PROGRAM sonotecCalibration
VAR_INPUT
	start : BOOL := FALSE;
	pumpA : BOOL := TRUE;
	setSpeedDuration : TIME := T#2M;
	runTestDuration : TIME := T#5M;
END_VAR
VAR_OUTPUT
	results : ARRAY[1..50] OF testResults;
END_VAR
VAR
	i : UINT := 0; // index
	n : UINT := 7;
	t : LREAL := 0.0;
	sp : ARRAY [1..50] OF LREAL := [80.0, 160.0, 240.0, 320.0, 400.0, 480.0, 560.0];
	//sp : ARRAY [1..50] OF LREAL := [51.0, 58.0, 64.0, 79.0, 97.0, 112.0, 128.0, 151.0, 210.0, 280.0, 335.0, 410.0, 480.0, 600.0];
	//sp : ARRAY [1..50] OF LREAL := [335.0, 410.0, 480.0, 600.0];
	setSpeed : SFCStepType;
	runTest : SFCStepType;
	recordTest : SFCStepType;
END_VAR

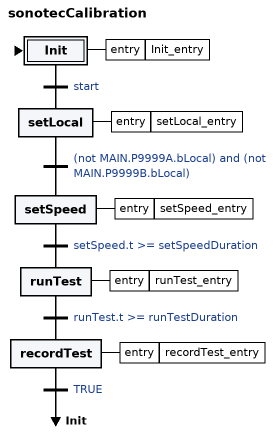
INITIAL_STEP Init:
    Init_entry(P1);  // entry action
END_STEP
TRANSITION FROM Init TO setLocal
    := start;
END_TRANSITION
STEP setLocal:
    setLocal_entry(P1);  // entry action
END_STEP
TRANSITION FROM setLocal TO setSpeed
    := (not MAIN.P9999A.bLocal) and (not MAIN.P9999B.bLocal);
END_TRANSITION
STEP setSpeed:
    setSpeed_entry(P1);  // entry action
END_STEP
TRANSITION FROM setSpeed TO runTest
    := setSpeed.t >= setSpeedDuration;
END_TRANSITION
STEP runTest:
    runTest_entry(P1);  // entry action
END_STEP
TRANSITION FROM runTest TO recordTest
    := runTest.t >= runTestDuration;
END_TRANSITION
STEP recordTest:
    recordTest_entry(P1);  // entry action
END_STEP
TRANSITION FROM recordTest TO Init
    := TRUE;
END_TRANSITION

ACTION setLocal_entry:
IF MAIN.P9999A.bLocal THEN
	MAIN.P9999A.nLocal_RQ := 0;  //put pump in remote
END_IF
IF MAIN.P9999B.bLocal THEN
	MAIN.P9999B.nLocal_RQ := 0;  //put pump in remote
END_IF
END_ACTION

ACTION runTest_entry:
MAIN.fbFQ9999A.resetRQ := TRUE;
MAIN.fbFQ9999B.resetRQ := TRUE;
MAIN.fbFQ9999C.resetRQ := TRUE;
END_ACTION

ACTION setSpeed_entry:
i := i + 1;
results[i].FQ9999A := 0.0;
results[i].FQ9999B := 0.0;
results[i].FQ9999C := 0.0;
results[i].FT9999Aavg := 0.0;
results[i].FT9999Bavg := 0.0;
results[i].FT9999Cavg := 0.0;
IF pumpA THEN
	results[i].P9999Arpm := sp[i];
	results[i].P9999Brpm := 0.0;
	MAIN.P9999A.nRun_RQ := 1; //start pump
	MAIN.P9999A.fSpeedSP_RQ := sp[i];
	MAIN.P9999B.nRun_RQ := 0; //stop pump
	MAIN.P9999B.fSpeedSP_RQ := 0.0;
ELSE
	results[i].P9999Arpm := 0.0;
	results[i].P9999Brpm := sp[i];
	MAIN.P9999A.nRun_RQ := 0; //stop pump
	MAIN.P9999A.fSpeedSP_RQ := 0.0;
	MAIN.P9999B.nRun_RQ := 1; //start pump
	MAIN.P9999B.fSpeedSP_RQ := sp[i];
END_IF
results[i].P9999Atubing := MAIN.P9999A.nTubeSize;
results[i].P9999Btubing := MAIN.P9999B.nTubeSize;
END_ACTION

ACTION recordTest_entry:
results[i].FQ9999A := MAIN.fbFQ9999A.total;
results[i].FQ9999B := MAIN.fbFQ9999B.total;
results[i].FQ9999C := MAIN.fbFQ9999C.total;
t := DWORD_TO_LREAL(TIME_TO_DWORD(runTestDuration))/1000.0/60.0;
results[i].FT9999Aavg := MAIN.fbFQ9999A.total/t;
results[i].FT9999Bavg := MAIN.fbFQ9999B.total/t;
results[i].FT9999Cavg := MAIN.fbFQ9999C.total/t;
END_ACTION

ACTION Init_entry:
IF i >= n THEN
	MAIN.P9999A.nRun_RQ := 0; //stop pump
	MAIN.P9999B.nRun_RQ := 0; //stop pump
	start := FALSE;
	i := 0;
END_IF
END_ACTION

END_PROGRAM

(* stored: Version 1.1.0.1, ProductVersion 3.1.0.36
   POU sonotecCalibration: Id {d8cace5d-4622-4721-8ad4-24bb2227c384}, SpecialFunc None
   Action setLocal_entry: Id {5f66cdec-b477-4613-901d-62d885f9dd8f}
   Action runTest_entry: Id {c408255e-879f-4b7c-a447-719d9549f349}
   Action setSpeed_entry: Id {d2f1a663-0229-4750-b307-3ef7969d2ce6}
   Action recordTest_entry: Id {ebcff068-10a2-4957-bb37-8ab7e3b316fc}
   Action Init_entry: Id {f93c3efd-ec5f-4afa-9577-f93e93fb7578} *)
